% RSLogix 500 project P10.RSS, saved by version 12.00.00.00 %
PROJECT "UNTITLED"    % processor: Bul.1763 MicroLogix 1100 Series B %

PROGRAM FILES
  LAD 2 "MAIN"  5 rungs
  LAD 3 "IO"  7 rungs
  LAD 4 "CONTROL"  5 rungs
  LAD 5 "ALARM"  8 rungs
  LAD 6 "ANALOG IO"  2 rungs

DATA FILES
  O0 OUTPUT  4 elements
  I1 INPUT  6 elements
  S2 STATUS  66 elements
  B3 BINARY  2 elements
  T4 TIMER  4 elements
  C5 COUNTER  1 elements
  R6 CONTROL  1 elements
  N7 INTEGER  3 elements
  F8 FLOAT  1 elements

LADDER 2 "MAIN"
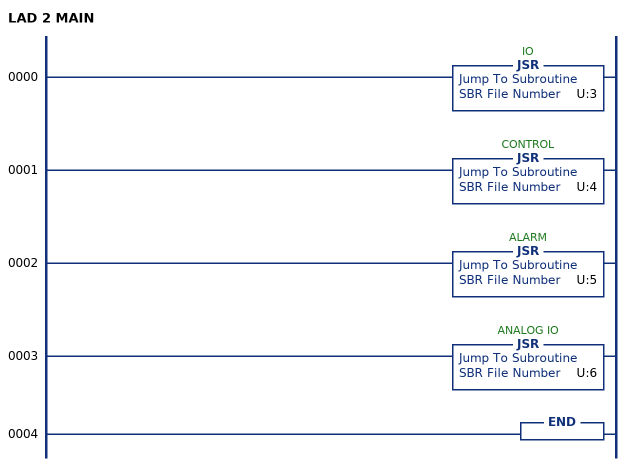
% Rung: 0 %
SOR JSR U:3 EOR
%   U:3  "IO" %
% Rung: 1 %
SOR JSR U:4 EOR
%   U:4  "CONTROL" %
% Rung: 2 %
SOR JSR U:5 EOR
%   U:5  "ALARM" %
% Rung: 3 %
SOR JSR U:6 EOR
%   U:6  "ANALOG IO" %
% Rung: 4 %
SOR END EOR

LADDER 3 "IO"
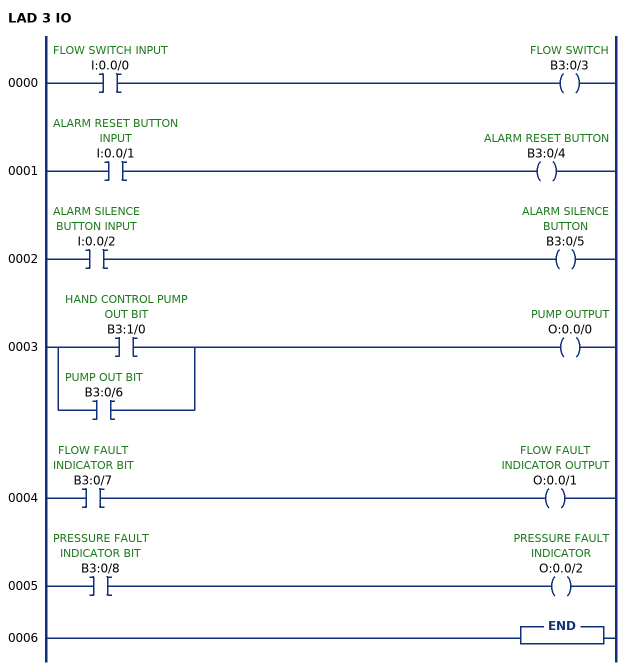
% Rung: 0 %
SOR XIC I:0.0/0 OTE B3:0/3 EOR
%   I:0.0/0  "FLOW SWITCH INPUT" %
%   B3:0/3  "FLOW SWITCH" %
% Rung: 1 %
SOR XIC I:0.0/1 OTE B3:0/4 EOR
%   I:0.0/1  "ALARM RESET BUTTON INPUT" %
%   B3:0/4  "ALARM RESET BUTTON" %
% Rung: 2 %
SOR XIC I:0.0/2 OTE B3:0/5 EOR
%   I:0.0/2  "ALARM SILENCE BUTTON INPUT" %
%   B3:0/5  "ALARM SILENCE BUTTON" %
% Rung: 3 %
SOR BST XIC B3:1/0 NXB XIC B3:0/6 BND OTE O:0.0/0 EOR
%   B3:1/0  "HAND CONTROL PUMP OUT BIT" %
%   B3:0/6  "PUMP OUT BIT" %
%   O:0.0/0  "PUMP OUTPUT" %
% Rung: 4 %
SOR XIC B3:0/7 OTE O:0.0/1 EOR
%   B3:0/7  "FLOW FAULT INDICATOR BIT" %
%   O:0.0/1  "FLOW FAULT INDICATOR OUTPUT" %
% Rung: 5 %
SOR XIC B3:0/8 OTE O:0.0/2 EOR
%   B3:0/8  "PRESSURE FAULT INDICATOR BIT" %
%   O:0.0/2  "PRESSURE FAULT INDICATOR" %
% Rung: 6 %
SOR END EOR

LADDER 4 "CONTROL"
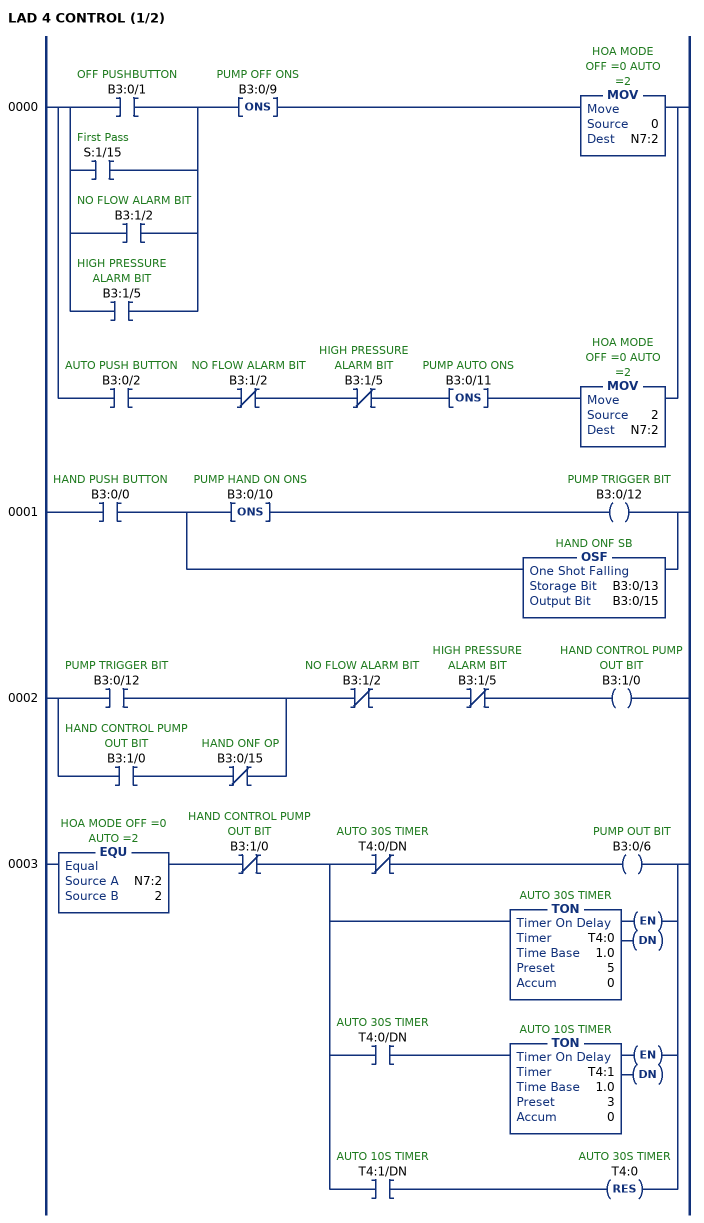
% Rung: 0 %
SOR BST BST XIC B3:0/1 NXB XIC S:1/15 NXB XIC B3:1/2 NXB XIC B3:1/5 BND ONS B3:0/9 MOV 0 N7:2 NXB XIC B3:0/2 XIO B3:1/2 XIO B3:1/5 ONS B3:0/11 MOV 2 N7:2 BND EOR
%   B3:0/1  "OFF PUSHBUTTON" %
%   S:1/15  "First Pass" %
%   B3:1/2  "NO FLOW ALARM BIT" %
%   B3:1/5  "HIGH PRESSURE ALARM BIT" %
%   B3:0/9  "PUMP OFF ONS" %
%   N7:2  "HOA MODE OFF =0 AUTO =2" %
%   B3:0/2  "AUTO PUSH BUTTON" %
%   B3:0/11  "PUMP AUTO ONS" %
% Rung: 1 %
SOR XIC B3:0/0 BST ONS B3:0/10 OTE B3:0/12 NXB OSF B3:0/13 B3:0/15 BND EOR
%   B3:0/0  "HAND PUSH BUTTON" %
%   B3:0/10  "PUMP HAND ON ONS" %
%   B3:0/12  "PUMP TRIGGER BIT" %
%   B3:0/13  "HAND ONF SB" %
%   B3:0/15  "HAND ONF OP" %
% Rung: 2 %
SOR BST XIC B3:0/12 NXB XIC B3:1/0 XIO B3:0/15 BND XIO B3:1/2 XIO B3:1/5 OTE B3:1/0 EOR
%   B3:0/12  "PUMP TRIGGER BIT" %
%   B3:1/0  "HAND CONTROL PUMP OUT BIT" %
%   B3:0/15  "HAND ONF OP" %
%   B3:1/2  "NO FLOW ALARM BIT" %
%   B3:1/5  "HIGH PRESSURE ALARM BIT" %
% Rung: 3 %
SOR EQU N7:2 2 XIO B3:1/0 BST XIO T4:0/DN OTE B3:0/6 NXB TON T4:0 1.0 5 0 NXB XIC T4:0/DN TON T4:1 1.0 3 0 NXB XIC T4:1/DN RES T4:0 BND EOR
%   N7:2  "HOA MODE OFF =0 AUTO =2" %
%   B3:1/0  "HAND CONTROL PUMP OUT BIT" %
%   T4:0  "AUTO 30S TIMER" %
%   B3:0/6  "PUMP OUT BIT" %
%   T4:1  "AUTO 10S TIMER" %

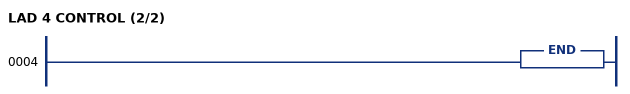
% Rung: 4 %
SOR END EOR

LADDER 5 "ALARM"
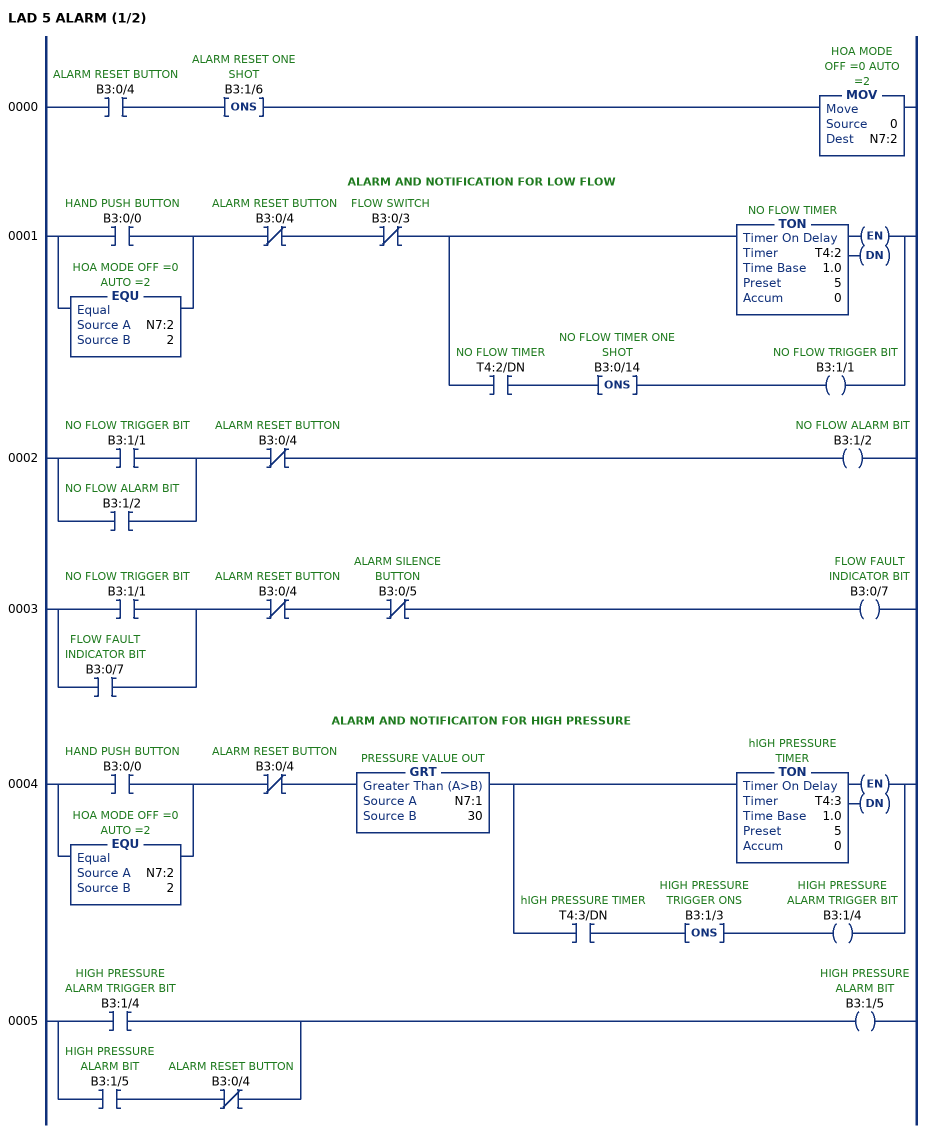
% Rung: 0 %
SOR XIC B3:0/4 ONS B3:1/6 MOV 0 N7:2 EOR
%   B3:0/4  "ALARM RESET BUTTON" %
%   B3:1/6  "ALARM RESET ONE SHOT" %
%   N7:2  "HOA MODE OFF =0 AUTO =2" %
% Rung: 1 %
% TITLE: ALARM AND NOTIFICATION FOR LOW FLOW %
SOR BST XIC B3:0/0 NXB EQU N7:2 2 BND XIO B3:0/4 XIO B3:0/3 BST TON T4:2 1.0 5 0 NXB XIC T4:2/DN ONS B3:0/14 OTE B3:1/1 BND EOR
%   B3:0/0  "HAND PUSH BUTTON" %
%   N7:2  "HOA MODE OFF =0 AUTO =2" %
%   B3:0/4  "ALARM RESET BUTTON" %
%   B3:0/3  "FLOW SWITCH" %
%   T4:2  "NO FLOW TIMER" %
%   B3:0/14  "NO FLOW TIMER ONE SHOT" %
%   B3:1/1  "NO FLOW TRIGGER BIT" %
% Rung: 2 %
SOR BST XIC B3:1/1 NXB XIC B3:1/2 BND XIO B3:0/4 OTE B3:1/2 EOR
%   B3:1/1  "NO FLOW TRIGGER BIT" %
%   B3:1/2  "NO FLOW ALARM BIT" %
%   B3:0/4  "ALARM RESET BUTTON" %
% Rung: 3 %
SOR BST XIC B3:1/1 NXB XIC B3:0/7 BND XIO B3:0/4 XIO B3:0/5 OTE B3:0/7 EOR
%   B3:1/1  "NO FLOW TRIGGER BIT" %
%   B3:0/7  "FLOW FAULT INDICATOR BIT" %
%   B3:0/4  "ALARM RESET BUTTON" %
%   B3:0/5  "ALARM SILENCE BUTTON" %
% Rung: 4 %
% TITLE: ALARM AND NOTIFICAITON FOR HIGH PRESSURE %
SOR BST XIC B3:0/0 NXB EQU N7:2 2 BND XIO B3:0/4 GRT N7:1 30 BST TON T4:3 1.0 5 0 NXB XIC T4:3/DN ONS B3:1/3 OTE B3:1/4 BND EOR
%   B3:0/0  "HAND PUSH BUTTON" %
%   N7:2  "HOA MODE OFF =0 AUTO =2" %
%   B3:0/4  "ALARM RESET BUTTON" %
%   N7:1  "PRESSURE VALUE OUT" %
%   T4:3  "hIGH PRESSURE TIMER" %
%   B3:1/3  "HIGH PRESSURE TRIGGER ONS" %
%   B3:1/4  "HIGH PRESSURE ALARM TRIGGER BIT" %
% Rung: 5 %
SOR BST XIC B3:1/4 NXB XIC B3:1/5 XIO B3:0/4 BND OTE B3:1/5 EOR
%   B3:1/4  "HIGH PRESSURE ALARM TRIGGER BIT" %
%   B3:1/5  "HIGH PRESSURE ALARM BIT" %
%   B3:0/4  "ALARM RESET BUTTON" %

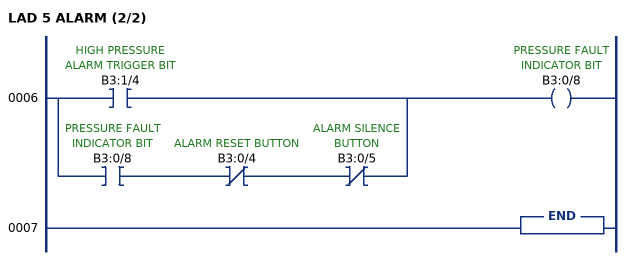
% Rung: 6 %
SOR BST XIC B3:1/4 NXB XIC B3:0/8 XIO B3:0/4 XIO B3:0/5 BND OTE B3:0/8 EOR
%   B3:1/4  "HIGH PRESSURE ALARM TRIGGER BIT" %
%   B3:0/8  "PRESSURE FAULT INDICATOR BIT" %
%   B3:0/4  "ALARM RESET BUTTON" %
%   B3:0/5  "ALARM SILENCE BUTTON" %
% Rung: 7 %
SOR END EOR

LADDER 6 "ANALOG IO"
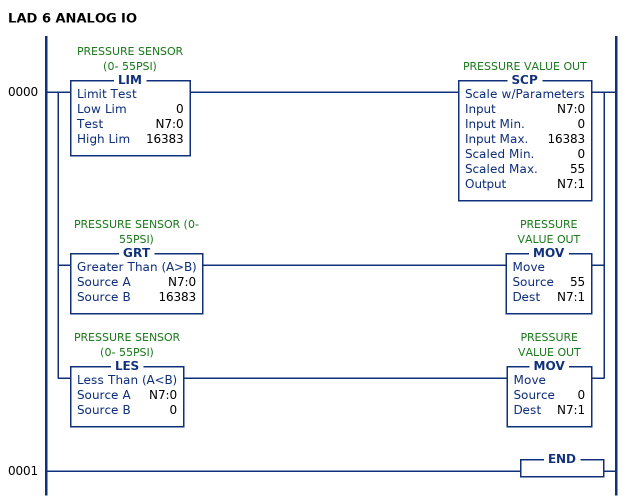
% Rung: 0 %
SOR BST LIM 0 N7:0 16383 SCP N7:0 0 16383 0 55 N7:1 NXB GRT N7:0 16383 MOV 55 N7:1 NXB LES N7:0 0 MOV 0 N7:1 BND EOR
%   N7:0  "PRESSURE SENSOR (0- 55PSI)" %
%   N7:1  "PRESSURE VALUE OUT" %
% Rung: 1 %
SOR END EOR

DATA TABLE (non-zero values as saved)
DATA T4
% .PRE .ACC %
% T4:0 % 5 0
% T4:1 % 3 0
% T4:2 % 5 0
% T4:3 % 5 0
